FUNCTION_BLOCK RfidHead_Test EXTENDS TcUnit.FB_TestSuite

ExecuteReadUid_ExpectUidAsStringStatusDone();

METHOD PRIVATE ExecuteReadUid_ExpectUidAsStringStatusDone
VAR_INST
    turckRfidHead : RfidHead(THIS^, T#1MS);
    sUId          : T_MaxString;
    _uid          : BOOL;
END_VAR
TcUnit.TEST('ExecuteReadUid_ExpectUidAsStringStatusDone');
turckRfidHead();

IF _uid THEN
    turckRfidHead.ReadUidMethod();
    _uid := FALSE;
END_IF

IF turckRfidHead.ReadUidTask.Done then
    sUId := turckRfidHead.sUId;
END_IF

TcUnit.TEST_FINISHED();
END_METHOD

END_FUNCTION_BLOCK

(* stored: Version 1.1.0.1, ProductVersion 3.1.4024.12
   POU RfidHead_Test: Id {a47ac61a-ee48-008c-0014-60e0cecfdf35}, SpecialFunc None
   Method ExecuteReadUid_ExpectUidAsStringStatusDone: Id {4cf9c36f-72dc-08b9-1fac-7b31252a268f} *)
